SUBAPPLICATION Uebung_054_AX (* DigitalInput_I1-_I4 auf DigitalOutput_Q1-_Q4, mit Plug and Socket *)
  (* Standard: 61499-2; Description: Copyright (c) 2026 Meisterschulen am Ostbahnhof This program and the accompanying materials are made available under the terms of the Eclipse Public License 2.0 which is available at https://www.eclipse.org/legal/epl-2.0/ SPDX-License-Identifier: EPL-2.0 *)
  (* Version 1.0, 2026-09-09, Franz Höpfinger, Meisterschulen am Ostbahnhof, initial API and implementation and/or initial documentation *)
  PACKAGE Uebungen;
  IMPORT logiBUS::io::DI::logiBUS_DI::Input_I1;
  IMPORT logiBUS::io::DI::logiBUS_DI::Input_I2;
  IMPORT logiBUS::io::DI::logiBUS_DI::Input_I3;
  IMPORT logiBUS::io::DI::logiBUS_DI::Input_I4;
  IMPORT logiBUS::io::DQ::logiBUS_DO::Output_Q1;
  IMPORT logiBUS::io::DQ::logiBUS_DO::Output_Q2;
  IMPORT logiBUS::io::DQ::logiBUS_DO::Output_Q3;
  IMPORT logiBUS::io::DQ::logiBUS_DO::Output_Q4;
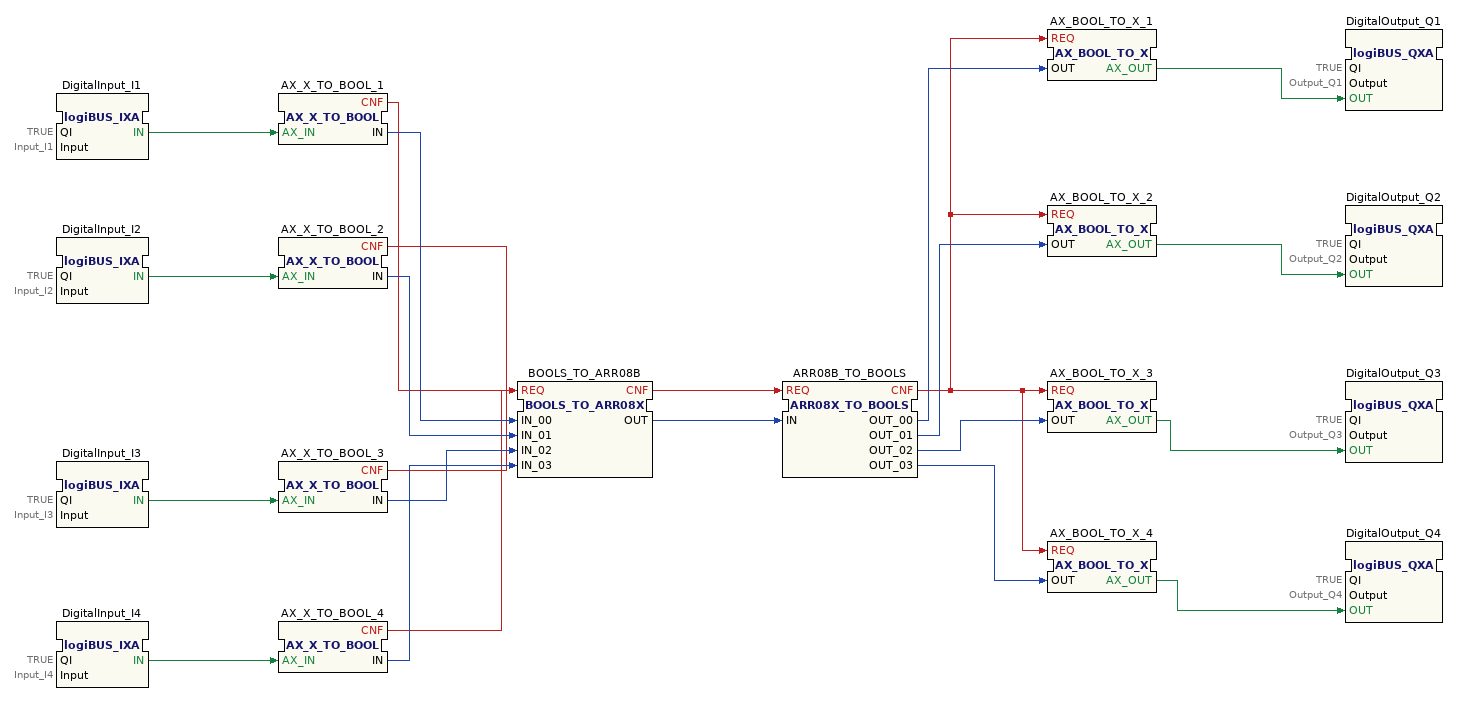
  FBS
    DigitalOutput_Q1 : logiBUS::io::DQ::logiBUS_QXA(QI := TRUE, Output := Output_Q1);
    DigitalInput_I1 : logiBUS::io::DI::logiBUS_IXA(QI := TRUE, Input := Input_I1);
    DigitalOutput_Q2 : logiBUS::io::DQ::logiBUS_QXA(QI := TRUE, Output := Output_Q2);
    DigitalInput_I2 : logiBUS::io::DI::logiBUS_IXA(QI := TRUE, Input := Input_I2);
    DigitalOutput_Q3 : logiBUS::io::DQ::logiBUS_QXA(QI := TRUE, Output := Output_Q3);
    DigitalInput_I3 : logiBUS::io::DI::logiBUS_IXA(QI := TRUE, Input := Input_I3);
    DigitalOutput_Q4 : logiBUS::io::DQ::logiBUS_QXA(QI := TRUE, Output := Output_Q4);
    DigitalInput_I4 : logiBUS::io::DI::logiBUS_IXA(QI := TRUE, Input := Input_I4);
    ARR08B_TO_BOOLS : logiBUS::utils::conversion::arr::forwarding::ARR08X_TO_BOOLS;
    BOOLS_TO_ARR08B : logiBUS::utils::conversion::arr::reversing::BOOLS_TO_ARR08X;
    AX_X_TO_BOOL_1 : adapter::conversion::unidirectional::AX_X_TO_BOOL;
    AX_X_TO_BOOL_2 : adapter::conversion::unidirectional::AX_X_TO_BOOL;
    AX_X_TO_BOOL_3 : adapter::conversion::unidirectional::AX_X_TO_BOOL;
    AX_X_TO_BOOL_4 : adapter::conversion::unidirectional::AX_X_TO_BOOL;
    AX_BOOL_TO_X_1 : adapter::conversion::unidirectional::AX_BOOL_TO_X;
    AX_BOOL_TO_X_2 : adapter::conversion::unidirectional::AX_BOOL_TO_X;
    AX_BOOL_TO_X_3 : adapter::conversion::unidirectional::AX_BOOL_TO_X;
    AX_BOOL_TO_X_4 : adapter::conversion::unidirectional::AX_BOOL_TO_X;
  END_FBS
  EVENT_CONNECTIONS
    BOOLS_TO_ARR08B.CNF TO ARR08B_TO_BOOLS.REQ;
    AX_X_TO_BOOL_1.CNF TO BOOLS_TO_ARR08B.REQ;
    AX_X_TO_BOOL_2.CNF TO BOOLS_TO_ARR08B.REQ;
    AX_X_TO_BOOL_3.CNF TO BOOLS_TO_ARR08B.REQ;
    AX_X_TO_BOOL_4.CNF TO BOOLS_TO_ARR08B.REQ;
    ARR08B_TO_BOOLS.CNF TO AX_BOOL_TO_X_1.REQ;
    ARR08B_TO_BOOLS.CNF TO AX_BOOL_TO_X_2.REQ;
    ARR08B_TO_BOOLS.CNF TO AX_BOOL_TO_X_3.REQ;
    ARR08B_TO_BOOLS.CNF TO AX_BOOL_TO_X_4.REQ;
  END_CONNECTIONS
  DATA_CONNECTIONS
    BOOLS_TO_ARR08B.OUT TO ARR08B_TO_BOOLS.IN;
    AX_X_TO_BOOL_1.IN TO BOOLS_TO_ARR08B.IN_00;
    AX_X_TO_BOOL_2.IN TO BOOLS_TO_ARR08B.IN_01;
    AX_X_TO_BOOL_3.IN TO BOOLS_TO_ARR08B.IN_02;
    AX_X_TO_BOOL_4.IN TO BOOLS_TO_ARR08B.IN_03;
    ARR08B_TO_BOOLS.OUT_00 TO AX_BOOL_TO_X_1.OUT;
    ARR08B_TO_BOOLS.OUT_01 TO AX_BOOL_TO_X_2.OUT;
    ARR08B_TO_BOOLS.OUT_02 TO AX_BOOL_TO_X_3.OUT;
    ARR08B_TO_BOOLS.OUT_03 TO AX_BOOL_TO_X_4.OUT;
  END_CONNECTIONS
  ADAPTER_CONNECTIONS
    DigitalInput_I1.IN TO AX_X_TO_BOOL_1.AX_IN;
    DigitalInput_I2.IN TO AX_X_TO_BOOL_2.AX_IN;
    DigitalInput_I3.IN TO AX_X_TO_BOOL_3.AX_IN;
    DigitalInput_I4.IN TO AX_X_TO_BOOL_4.AX_IN;
    AX_BOOL_TO_X_1.AX_OUT TO DigitalOutput_Q1.OUT;
    AX_BOOL_TO_X_2.AX_OUT TO DigitalOutput_Q2.OUT;
    AX_BOOL_TO_X_3.AX_OUT TO DigitalOutput_Q3.OUT;
    AX_BOOL_TO_X_4.AX_OUT TO DigitalOutput_Q4.OUT;
  END_CONNECTIONS
END_SUBAPPLICATION
